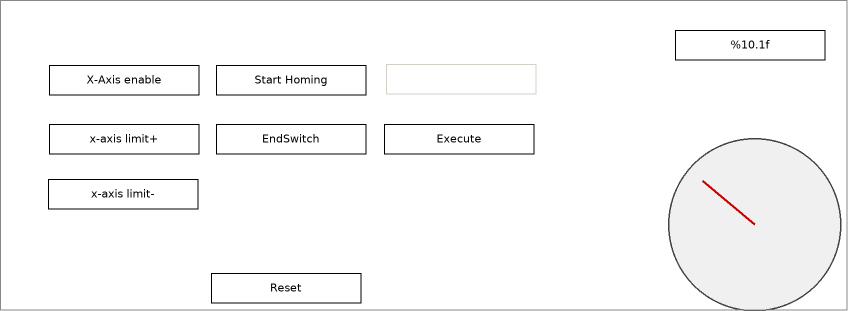
VISUALIZATION testStepperVisu  // 848x311
    Rectangle (49,65 150x30), "X-Axis enable"
        toggle GVL_AxisCtr.bXAxisEnable
    RoundedRectangle (49,124 150x30), "x-axis limit+", colour toggle: GVL_IO.I_bXAxisLimitSwPos
        toggle GVL_IO.I_bXAxisLimitSwPos
    RoundedRectangle (48,179 150x30), "x-axis limit-", colour toggle: GVL_IO.I_bXAxisLimitSwNeg
        toggle GVL_IO.I_bXAxisLimitSwNeg
    Rectangle (675,30 150x30), "%10.1f", text variable: GVL_NC.stXAxis.NcToPlc.ActPos
    Rectangle (384,124 150x30), "Execute"
        tap movements.ExecuteMovement
    Rectangle (216,65 150x30), "Start Homing"
        tap POUNCPowerOn.StartHoming
    Rectangle (216,124 150x30), "EndSwitch"
        toggle POUNCPowerOn.endSW
    Rectangle (211,273 150x30), "Reset"
        tap POUNCPowerOn.reset
    Meter90 (661,138 187x173), value: movements.PositionToDegree_0.Deg, style: Meter-Meter90-Gray, scale format: %.1f, scale -45..45
    Textfield (386,64 150x30), text variable: movements.Command_to_Action_0.inputString
        OnMouseDown: write the text variable via Default
END_VISUALIZATION

(* stored: Version 1.1.0.1, ProductVersion 3.1.4024.3
   Visu testStepperVisu: Id {874346f2-d8fd-4506-a2c5-a06924bc3234} *)
